(* IEC 61131-3 sources: horner-cscape-mcp/artifacts/projects/Fail_Syntax_Location_Proj/pous, 1 file *)

(* ---- POU_SyntaxError.st ---- *)
PROGRAM POU_SyntaxError
VAR
    Speed : INT := 100;
END_VAR

IF Speed > 50 THEN
    Speed := 50;
(* Intentional syntax error: unclosed IF missing END_IF *)

END_PROGRAM
